{attribute 'qualified_only'}
VAR_GLOBAL
    {attribute 'pytmc' := 'pv: SL2K4:SCATTER:MMS:BOTTOM'}
    M1 : DUT_MotionStage := (nEnableMode:=ENUM_StageEnableMode.DURING_MOTION, bPowerSelf:=TRUE);

	{attribute 'pytmc' := 'pv: SL2K4:SCATTER:MMS:NORTH'}
    M2 : DUT_MotionStage := (nEnableMode:=ENUM_StageEnableMode.DURING_MOTION, bPowerSelf:=TRUE);

    {attribute 'pytmc' := 'pv: SL2K4:SCATTER:MMS:TOP'}
    M3 : DUT_MotionStage := (nEnableMode:=ENUM_StageEnableMode.DURING_MOTION, bPowerSelf:=TRUE);

	{attribute 'pytmc' := 'pv: SL2K4:SCATTER:MMS:SOUTH'}
    M4 : DUT_MotionStage := (nEnableMode:=ENUM_StageEnableMode.DURING_MOTION, bPowerSelf:=TRUE);
END_VAR

(* stored: Version 1.1.0.1, ProductVersion 3.1.4024.12
   GVL GVL: Id {6f81f5f7-0a84-4a54-8d7d-5984f3eae6b9} *)
